GLOBALCONSTANTS AID_SG (* Scaled graphic object attribute ids *)
  (* Standard: 61499-1; Description: Copyright (c) 2023 HR Agrartechnik GmbH This program and the accompanying materials are made available under the terms of the Eclipse Public License 2.0 which is available at https://www.eclipse.org/legal/epl-2.0/ SPDX-License-Identifier: EPL-2.0 *)
  (* Version 1.0, 2026-06-20, Franz Höpfinger, HR Agrartechnik GmbH *)
  PACKAGE isobus::UT::Q::const::AID;
  VAR_GLOBAL CONSTANT
    WIDTH : USINT := USINT#1; (* 1: AID_SG_WIDTH - Width in pixels. *)
    HEIGHT : USINT := USINT#2; (* 2: AID_SG_HEIGHT - Height in pixels. *)
    SCALE_TYPE : USINT := USINT#3; (* 3: AID_SG_SCALE_TYPE - Bits 0-2: Scaling Value (0=no scale, 1=scale to width, 2=scale to height, *)
    OPTIONS : USINT := USINT#4; (* 4: AID_SG_OPTIONS - Bitmask: Bit 0=Flashing. *)
    VALUE : USINT := USINT#5; (* 5: AID_SG_VALUE - [5] Read-only attribute. Object ID of referenced graphic object. Runtime mod via F.22. *)
  END_VAR
END_GLOBALCONSTANTS
